FUNCTION_BLOCK FB_DiagnosticMessageFlagsParser_Test EXTENDS TcUnit.FB_TestSuite

WhenInfoMessageExpectInfoMessageGlobalTimestampAndZeroParameters();
WhenWarningMessageExpectWarningMessageLocalTimestampAndTwoParameters();
WhenErrorMessageExpectErrorMessageLocalTimestampAndFourParameters();
WhenReservedForFutureUseMessageExpectReservedForFutureUseMessageLocalTimestampAnd33Parameters();

METHOD PRIVATE WhenErrorMessageExpectErrorMessageLocalTimestampAndFourParameters
VAR
    fbDiagnosticMessageFlagsParser : FB_DiagnosticMessageFlagsParser;
    stFlags : ST_FLAGS;

    // @TEST-FIXTURE ErrorMessage
    cnFlagsBufferByte1_ErrorMessage : BYTE := 2#0001_0010; // Error message and local time stamp
    cnFlagsBufferByte2_ErrorMessage : BYTE := 2#0000_0100; // Four parameters in the diagnosis message
    canFlagsBuffer_ErrorMessage : ARRAY[1..2] OF BYTE := [cnFlagsBufferByte1_ErrorMessage, 
                                                          cnFlagsBufferByte2_ErrorMessage];
    // @TEST-RESULT ErrorMessage
    ceFlags_DiagnosisTypeErrorMessage : E_DIAGNOSISTYPE := E_DIAGNOSISTYPE.ErrorMessage;
    ceFlags_TimeStampTypeLocal : E_TIMESTAMPTYPE := E_TIMESTAMPTYPE.Local;
    cnFlags_NumberOfParametersInDiagnosisMessageFour : USINT := 4;
END_VAR
TEST('WhenErrorMessageExpectErrorMessageLocalTimestampAndFourParameters');

// @TEST-RUN ErrorMessage
fbDiagnosticMessageFlagsParser(anFlagsBuffer := canFlagsBuffer_ErrorMessage,
                               stFlags => stFlags);

// @TEST-ASSERT ErrorMessage
AssertEquals(Expected := ceFlags_DiagnosisTypeErrorMessage,
             Actual := stFlags.eDiagnosisType,
             'Test $'Error message$' failed at $'diagnosis type$'');
AssertEquals(Expected := ceFlags_TimeStampTypeLocal,
             Actual := stFlags.eTimeStampType,
             'Test $'Error message$' failed at $'timestamp type$'');
AssertEquals(Expected := cnFlags_NumberOfParametersInDiagnosisMessageFour,
             Actual := stFlags.nNumberOfParametersInDiagnosisMessage,
             'Test $'Error message$' failed at $'number of parameters$'');

TEST_FINISHED();
END_METHOD

METHOD PRIVATE WhenInfoMessageExpectInfoMessageGlobalTimestampAndZeroParameters
VAR
    fbDiagnosticMessageFlagsParser : FB_DiagnosticMessageFlagsParser;
    stFlags : ST_FLAGS;

    // @TEST-FIXTURE InfoMessage
    cnFlagsBufferByte1_InfoMessage : BYTE := 2#0000_0000; // Info message and global time stamp
    cnFlagsBufferByte2_InfoMessage : BYTE := 2#0000_0000; // Zero parameters in the diagnosis message
    canFlagsBuffer_InfoMessage : ARRAY[1..2] OF BYTE := [cnFlagsBufferByte1_InfoMessage, 
                                                         cnFlagsBufferByte2_InfoMessage];
    // @TEST-RESULT InfoMessage
    ceFlags_DiagnosisTypeInfoMessage : E_DIAGNOSISTYPE := E_DIAGNOSISTYPE.InfoMessage;
    ceFlags_TimeStampTypeGlobal : E_TIMESTAMPTYPE := E_TIMESTAMPTYPE.Global;
    cnFlags_NumberOfParametersInDiagnosisMessageZero : USINT := 0;
END_VAR
TEST('WhenInfoMessageExpectInfoMessageGlobalTimestampAndZeroParameters');

// @TEST-RUN
fbDiagnosticMessageFlagsParser(anFlagsBuffer := canFlagsBuffer_InfoMessage,
                               stFlags => stFlags);

// @TEST-ASSERT
AssertEquals(Expected := ceFlags_DiagnosisTypeInfoMessage,
             Actual := stFlags.eDiagnosisType,
             'Test $'Info message$' failed at $'diagnosis type$'');
AssertEquals(Expected := ceFlags_TimeStampTypeGlobal,
             Actual := stFlags.eTimeStampType,
             'Test $'Info message$' failed at $'timestamp type$'');
AssertEquals(Expected := cnFlags_NumberOfParametersInDiagnosisMessageZero,
             Actual := stFlags.nNumberOfParametersInDiagnosisMessage,
             'Test $'Info message$' failed at $'number of parameters$'');

TEST_FINISHED();
END_METHOD

METHOD PRIVATE WhenReservedForFutureUseMessageExpectReservedForFutureUseMessageLocalTimestampAnd33Parameters
VAR
    fbDiagnosticMessageFlagsParser : FB_DiagnosticMessageFlagsParser;
    stFlags : ST_FLAGS;

    // @TEST-FIXTURE ReservedForFutureUseMessage
    cnFlagsBufferByte1_ReservedForFutureUseMessage : BYTE := 2#0001_0011; // ReservedForFutureUse message and local time stamp
    cnFlagsBufferByte2_ReservedForFutureUseMessage : BYTE := 2#0010_0001; // 33 parameters in the diagnosis message
    canFlagsBuffer_ReservedForFutureUseMessage : ARRAY[1..2] OF BYTE := [cnFlagsBufferByte1_ReservedForFutureUseMessage, 
                                                                         cnFlagsBufferByte2_ReservedForFutureUseMessage];
    // @TEST-RESULT ReservedForFutureUseMessage
    ceFlags_DiagnosisTypeReservedForFutureUseMessage : E_DIAGNOSISTYPE := E_DIAGNOSISTYPE.Unspecified;
    cnFlags_NumberOfParametersInDiagnosisMessage33 : USINT := 33;
    ceFlags_TimeStampTypeLocal : E_TIMESTAMPTYPE := E_TIMESTAMPTYPE.Local;
END_VAR
TEST('WhenReservedForFutureUseMessageExpectReservedForFutureUseMessageLocalTimestampAnd33Parameters');

// @TEST-RUN ReservedForFutureUseMessage
fbDiagnosticMessageFlagsParser(anFlagsBuffer := canFlagsBuffer_ReservedForFutureUseMessage,
                               stFlags => stFlags);

// @TEST-ASSERT ReservedForFutureUseMessage
AssertEquals(Expected := ceFlags_DiagnosisTypeReservedForFutureUseMessage,
             Actual := stFlags.eDiagnosisType,
             'Test $'Reserved for future use message$' failed at $'diagnosis type$'');
AssertEquals(Expected := ceFlags_TimeStampTypeLocal,
             Actual := stFlags.eTimeStampType,
             'Test $'Reserved for future use message$' failed at $'timestamp type$'');
AssertEquals(Expected := cnFlags_NumberOfParametersInDiagnosisMessage33,
             Actual := stFlags.nNumberOfParametersInDiagnosisMessage,
             'Test $'Reserved for future use message$' failed at $'number of parameters$'');

TEST_FINISHED();
END_METHOD

METHOD PRIVATE WhenWarningMessageExpectWarningMessageLocalTimestampAndTwoParameters
VAR
    fbDiagnosticMessageFlagsParser : FB_DiagnosticMessageFlagsParser;
    stFlags : ST_FLAGS;

    // @TEST-FIXTURE WarningMessage
    cnFlagsBufferByte1_WarningMessage : BYTE := 2#0001_0001; // Warning message and local time stamp
    cnFlagsBufferByte2_WarningMessage : BYTE := 2#0000_0010; // Two parameters in the diagnosis message
    canFlagsBuffer_WarningMessage : ARRAY[1..2] OF BYTE := [cnFlagsBufferByte1_WarningMessage, 
                                                            cnFlagsBufferByte2_WarningMessage];
    // @TEST-RESULT WarningMessage
    ceFlags_DiagnosisTypeWarningMessage : E_DIAGNOSISTYPE := E_DIAGNOSISTYPE.WarningMessage;
    ceFlags_TimeStampTypeLocal : E_TIMESTAMPTYPE := E_TIMESTAMPTYPE.Local;
    cnFlags_NumberOfParametersInDiagnosisMessageTwo : USINT := 2;
END_VAR
TEST('WhenWarningMessageExpectWarningMessageLocalTimestampAndTwoParameters');

// @TEST-RUN WarningMessage
fbDiagnosticMessageFlagsParser(anFlagsBuffer := canFlagsBuffer_WarningMessage,
                               stFlags => stFlags);

// @TEST-ASSERT WarningMessage
AssertEquals(Expected := ceFlags_DiagnosisTypeWarningMessage,
             Actual := stFlags.eDiagnosisType,
             'Test $'Warning message$' failed at $'diagnosis type$'');
AssertEquals(Expected := ceFlags_TimeStampTypeLocal,
             Actual := stFlags.eTimeStampType,
             'Test $'Warning message$' failed at $'timestamp type$'');
AssertEquals(Expected := cnFlags_NumberOfParametersInDiagnosisMessageTwo,
             Actual := stFlags.nNumberOfParametersInDiagnosisMessage,
             'Test $'Warning message$' failed at $'number of parameters$'');

TEST_FINISHED();
END_METHOD

END_FUNCTION_BLOCK

(* stored: Version 1.1.0.1
   POU FB_DiagnosticMessageFlagsParser_Test: Id {2c0e6355-6af7-46b0-9fcf-479aaac3c4bc}, SpecialFunc None
   Method WhenErrorMessageExpectErrorMessageLocalTimestampAndFourParameters: Id {9a9c4539-6094-4180-9da4-a22f03bc41c6}
   Method WhenInfoMessageExpectInfoMessageGlobalTimestampAndZeroParameters: Id {bb46ac41-02ed-40ed-a816-83fb6980e06d}
   Method WhenReservedForFutureUseMessageExpectReservedForFutureUseMessageLocalTimestampAnd33Parameters: Id {6be770b4-b74f-46a4-964f-1c71e63b7446}
   Method WhenWarningMessageExpectWarningMessageLocalTimestampAndTwoParameters: Id {da79b77f-b650-455b-a807-dff9ec60e1b5} *)
